{attribute addProperty BoxType "KL8610-0001"}
{attribute addProperty Id "KL8601_1KL_B0A8062F00KL8601_2KL_B0A8062F00"}
{attribute addProperty CRC "1323789305"}
{attribute addProperty SizeInBites "0"}
{attribute addProperty SizeInBytes "0"}
TYPE KL_4EE76BF9 :
STRUCT
	{attribute addProperty Name "KL8601_1"}
	KL8601_1 : KL_B0A8062F;
	{attribute addProperty Name "KL8601_2"}
	KL8601_2 : KL_B0A8062F;
END_STRUCT
END_TYPE

(* stored: Version 1.2.0.0, ProductVersion 3.1.4024.9
   DUT KL_4EE76BF9: Id {b3db963d-b2c2-43b9-b413-87051dfd5514} *)
